// TIA Portal V19 export
DATA_BLOCK "Letter_A"   // DB4
{ S7_Optimized_Access := 'TRUE' }
// stored: MemoryReserve 100
   VAR
      Coordinates : Array[0..5] of "XYZ_Coordinates";
   END_VAR
BEGIN
   Coordinates[0..2].X := 1.0;
   Coordinates[0..2].Y := 2.0;
   Coordinates[0..2].Z := 3.0;
END_DATA_BLOCK
